Fanuc KAREL source: NC0080.compact.KL

PROGRAM NC0080
%STACKSIZE=65535
%PRIORITY=65535
%NOLOCKGROUP
ROUTINE R FROM NC0080
ROUTINE R
VAR
S1 : INTEGER
BEGIN
S1=1
WHILE (S1 < 2) DO
WHILE (S1 < 2) DO
WHILE (S1 < 2) DO
WHILE (S1 < 2) DO
WHILE (S1 < 2) DO
WHILE (S1 < 2) DO
WHILE (S1 < 2) DO
WHILE (S1 < 2) DO
WHILE (S1 < 2) DO
WHILE (S1 < 2) DO
WHILE (S1 < 2) DO
WHILE (S1 < 2) DO
WHILE (S1 < 2) DO
WHILE (S1 < 2) DO
WHILE (S1 < 2) DO
WHILE (S1 < 2) DO
WHILE (S1 < 2) DO
WHILE (S1 < 2) DO
S1=(S1 + 1)
ENDWHILE
ENDWHILE
ENDWHILE
ENDWHILE
ENDWHILE
ENDWHILE
ENDWHILE
ENDWHILE
ENDWHILE
ENDWHILE
ENDWHILE
ENDWHILE
ENDWHILE
ENDWHILE
ENDWHILE
ENDWHILE
ENDWHILE
ENDWHILE
END R
BEGIN
R
END NC0080
